// TIA Portal V19 export
FUNCTION_BLOCK "1200Comm"   // FB3, LAD
TITLE = I Device exchange of data with the S7-1200
{ S7_Optimized_Access := 'TRUE' }
// stored: MemoryReserve 100, SetENOAutomatically false
BEGIN

REGION Network 1: Pass light data to the 1200
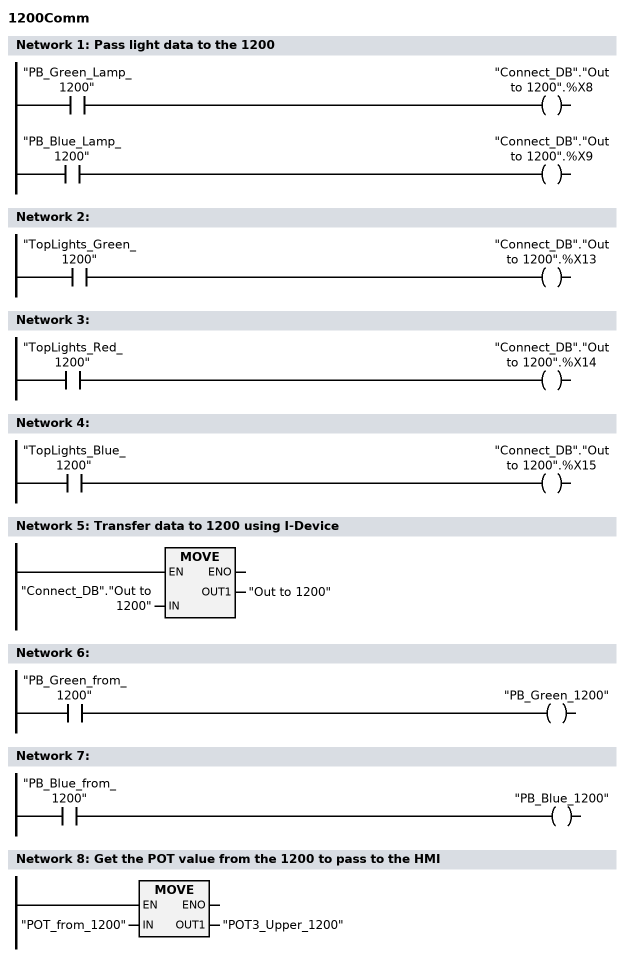
   RUNG wire#powerrail
      Contact( "PB_Green_Lamp_1200" )
      Coil( "Connect_DB"."Out to 1200".%X8 )
   END_RUNG
   RUNG wire#powerrail
      Contact( "PB_Blue_Lamp_1200" )
      Coil( "Connect_DB"."Out to 1200".%X9 )
   END_RUNG
   // the same network as SCL:
   "Connect_DB"."Out to 1200".%X8 := "PB_Green_Lamp_1200";
   "Connect_DB"."Out to 1200".%X9 := "PB_Blue_Lamp_1200";
END_REGION

REGION Network 2
   RUNG wire#powerrail
      Contact( "TopLights_Green_1200" )
      Coil( "Connect_DB"."Out to 1200".%X13 )
   END_RUNG
   // the same network as SCL:
   "Connect_DB"."Out to 1200".%X13 := "TopLights_Green_1200";
END_REGION

REGION Network 3
   RUNG wire#powerrail
      Contact( "TopLights_Red_1200" )
      Coil( "Connect_DB"."Out to 1200".%X14 )
   END_RUNG
   // the same network as SCL:
   "Connect_DB"."Out to 1200".%X14 := "TopLights_Red_1200";
END_REGION

REGION Network 4
   RUNG wire#powerrail
      Contact( "TopLights_Blue_1200" )
      Coil( "Connect_DB"."Out to 1200".%X15 )
   END_RUNG
   // the same network as SCL:
   "Connect_DB"."Out to 1200".%X15 := "TopLights_Blue_1200";
END_REGION

REGION Network 5: Transfer data to 1200 using I-Device
   RUNG wire#powerrail
      Move(in := "Connect_DB"."Out to 1200", out1 => "Out to 1200")
   END_RUNG
   // the same network as SCL:
   "Out to 1200" := "Connect_DB"."Out to 1200";
END_REGION

REGION Network 6
   RUNG wire#powerrail
      Contact( "PB_Green_from_1200" )
      Coil( "PB_Green_1200" )
   END_RUNG
   // the same network as SCL:
   "PB_Green_1200" := "PB_Green_from_1200";
END_REGION

REGION Network 7
   RUNG wire#powerrail
      Contact( "PB_Blue_from_1200" )
      Coil( "PB_Blue_1200" )
   END_RUNG
   // the same network as SCL:
   "PB_Blue_1200" := "PB_Blue_from_1200";
END_REGION

REGION Network 8: Get the POT value from the 1200 to pass to the HMI
   RUNG wire#powerrail
      Move(in := "POT_from_1200", out1 => "POT3_Upper_1200")
   END_RUNG
   // the same network as SCL:
   "POT3_Upper_1200" := "POT_from_1200";
END_REGION
END_FUNCTION_BLOCK
